PROGRAM MAIN
VAR
END_VAR

END_PROGRAM

(* stored: Version 1.1.0.1
   POU MAIN: Id {74cf7d8f-31c3-4dfc-b90c-a054170cc2a4} *)
